(*
SPDX-FileCopyrightText: Â© 2026 Oleksandr Tiutyk <trofimich@gmail.com>
SPDX-License-Identifier: MIT
License: https://opensource.org/license/mit
*)

(*!
<summary>Contract for analog signal scaling and engineering unit conversion.</summary>
<description>
Converts raw ADC/DAC values to and from engineering unit LREAL representations.
</description>
*)

INTERFACE IAnalogValueConverter EXTENDS TOF_Core.IObject

(*!
<summary>Converts an engineering unit value to raw hardware representation.</summary>
<param name="analogValue">Engineering unit analog value.</param>
<param name="rawValueType">Target raw data representation.</param>
*)
METHOD ConvertAnalogValueToRawValue : RAW_ANALOG_VALUE
VAR_INPUT
	analogValue : LREAL;
	rawValueType : RAW_ANALOG_VALUE_TYPE;
END_VAR
END_METHOD

(*!
<summary>Converts raw hardware representation to an engineering unit value.</summary>
<param name="rawValue">Raw process value union.</param>
<param name="rawValueType">Source raw data representation.</param>
*)
METHOD ConvertRawValueToAnalogValue : LREAL
VAR_INPUT
	rawValue : RAW_ANALOG_VALUE;
	rawValueType : RAW_ANALOG_VALUE_TYPE;
END_VAR
END_METHOD

END_INTERFACE

(* stored: Version 1.1.0.1
   Itf IAnalogValueConverter: Id {996c28a6-ed43-435b-bd2d-4a48e125454f}
   Method ConvertAnalogValueToRawValue: Id {7b9f8ba6-8d64-4125-89ee-b6b6b6ab7033}
   Method ConvertRawValueToAnalogValue: Id {8ee92332-8449-42df-aea2-819ba3290c45} *)
